INTERFACE I_SMPTE_TimeController

METHOD Cycle : BOOL
VAR_INPUT
END_VAR
END_METHOD

// Will pause the time
METHOD Pause : BOOL
VAR_INPUT
	bExecute : BOOL;
END_VAR
END_METHOD

PROPERTY Paused : BOOL
GET
END_GET
END_PROPERTY

// Starts the time
METHOD Play : BOOL
VAR_INPUT
	bExecute : BOOL;
END_VAR
END_METHOD

PROPERTY Playing : BOOL
GET
END_GET
END_PROPERTY

// Resets the time
METHOD Reset : BOOL
VAR_INPUT
	bExecute : BOOL;
END_VAR
END_METHOD

// Will stop the time and reset to 00:00:00:00
METHOD Stop : BOOL
VAR_INPUT
	bExecute : BOOL;
END_VAR
END_METHOD

PROPERTY Stopped : BOOL
GET
END_GET
END_PROPERTY

// Returns the SMPTE_Sender_TimeStruct
PROPERTY TimeStruct : REFERENCE TO ST_SMPTE_TimeStruct;
GET
END_GET
END_PROPERTY

END_INTERFACE

(* stored: Version 1.1.0.1, ProductVersion 3.1.4024.12
   Itf I_SMPTE_TimeController: Id {a810304c-d5d0-495a-ae08-e61f0e71c0b0}
   Folder Public: Id {cb6fe0d9-0e20-4f3e-a7b6-4cfb726f81f8}
   Method Cycle: Id {55fd8665-20f5-4253-8b18-37d1a4d16b96}
   Method Pause: Id {69b1702a-0797-4e36-bc96-01b210c9bc4a}
   Property Paused: Id {8aeba0db-db0f-4613-890e-d91813ba6553}
   Get Get: Id {727a3d17-5dad-4048-906e-6dcde70d97bc}
   Method Play: Id {2ba88ade-d166-4063-8ede-cd22dfce61ca}
   Property Playing: Id {1cc8b953-eb51-4c82-bc38-858549a6cce2}
   Get Get: Id {7ca3aceb-4894-470b-a67b-94676098a162}
   Method Reset: Id {28ae49f6-0f8a-4f79-9428-0a70fb3f6523}
   Method Stop: Id {c47c79bd-dd6a-4839-a5ec-0ca1698e0ea5}
   Property Stopped: Id {2932507c-8a2a-4151-8d5e-1a922b4882e4}
   Get Get: Id {703663ed-26a3-4e32-8c8f-6b78da24d556}
   Property TimeStruct: Id {844ce3d6-1d05-47f7-8dd9-51d704786b17}
   Get Get: Id {7fbae9f9-b418-4807-8db5-949148fba8b3} *)
